PROGRAM P_Demo_FB_DMXDiscMute
VAR
    fbDiscMute        : FB_DMXDiscMute;               // 置位设备 mute 标志
    stDmxCmdBuffer    : ST_DMXCommandBuffer;          // 与通讯 FB 共用
    wTargetManufId    : WORD := 16#4241;              // 目标灯具厂商 ID
    dwTargetDeviceId  : DWORD := 16#12131415;         // 目标灯具设备 ID
    byTargetPort      : BYTE := 0;                    // 根设备通道 0
    bDoMute           : BOOL := FALSE;                // 在线给一次上升沿触发
    bBusy             : BOOL;
    bError            : BOOL;
    udiErrId          : UDINT;
    wCtrlField        : WORD;                         // 设备返回的控制字段
END_VAR

// ============================================================
// Tc2_DMX.FB_DMXDiscMute 演示程序
// ============================================================
// 场景：自写定制发现流程（如只在某 UID 子区间搜索）时，手动 mute 已确认设备以缩小搜索范围。
// 价值：把 RDM 发现协议中的 mute 步骤暴露为单独 FB，给需要自定义发现策略的用户精细控制权。
// 验证：给 bDoMute 一次上升沿 -> bBusy 短暂 TRUE -> 回 FALSE 后 wCtrlField 有值；之后对同一设备发 FB_DMXDiscUniqueBranch 应不再得到响应（已被 mute）。
// 验证步骤：
//   1. 右键 PLC 项目下 POUs 文件夹 → Add → Existing Item → 选本 .TcPOU 文件
//   2. 引用 Tc2_DMX；同项目里放一个 FB_EL6851CommunicationEx 实例并共用 stDmxCmdBuffer（非 CycleMode）
//   3. 编译 → 登录 → 运行；按上方『验证』行在线给上升沿观察
// ============================================================

fbDiscMute(
    bStart                     := bDoMute,
    wDestinationManufacturerId := wTargetManufId,
    dwDestinationDeviceId      := dwTargetDeviceId,
    byPortId                   := byTargetPort,
    dwOptions                  := 0,
    stCommandBuffer            := stDmxCmdBuffer,
    bBusy                      => bBusy,
    bError                     => bError,
    udiErrorId                 => udiErrId,
    wControlField              => wCtrlField
);

END_PROGRAM

(* stored: Version 1.1.0.1, ProductVersion 3.1.4024.5
   POU P_Demo_FB_DMXDiscMute: Id {854c123b-7889-5727-b841-be37d4fe319f}, SpecialFunc None *)
